FUNCTION_BLOCK AUI_MUX_7 (* Event multiplexer with AUI adapter output instead of plain EO+K (generic FB) *)
  (* Standard: 61499-1 Annex A; Description: Copyright (c) 2017, 2025 fortiss GmbH, HR Agrartechnik GmbH This program and the accompanying materials are made available under the terms of the Eclipse Public License 2.0 which is available at https://www.eclipse.org/legal/epl-2.0/ SPDX-License-Identifier: EPL-2.0 *)
  (* Version 1.0, 2026-09-10, Franz Höpfinger, HR Agrartechnik GmbH, AUI adapter variant of E_MUX_7 *)
  PACKAGE adapter::events::unidirectional;
  {SET_ATTRIBUTE(eclipse4diac::core::GenericClassName, 'GEN_AUI_MUX')}
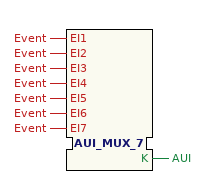
  EVENT_INPUT
    EI1; (* Event to multiplex, K=0 *)
    EI2; (* Event to multiplex, K=1 *)
    EI3; (* Event to multiplex, K=2 *)
    EI4; (* Event to multiplex, K=3 *)
    EI5; (* Event to multiplex, K=4 *)
    EI6; (* Event to multiplex, K=5 *)
    EI7; (* Event to multiplex, K=6 *)
  END_EVENT
  PLUGS
    K : adapter::types::unidirectional::AUI; (* Event index *)
  END_PLUGS
END_FUNCTION_BLOCK
